TYPE ST_Triggers :
STRUCT
	Left: ST_Trigger;
	Right: ST_Trigger;
END_STRUCT
END_TYPE

(* stored: Version 1.1.0.1
   DUT ST_Triggers: Id {23fe38f5-1749-4c16-9421-9a5256c84443} *)
